TYPE ST_IOInputSimul :
STRUCT
	IxAru :BOOL;
END_STRUCT
END_TYPE

(* stored: Version 1.1.0.1, ProductVersion 3.1.4020.6
   DUT ST_IOInputSimul: Id {0eeda127-7f03-4f22-8390-7883b0f0db7e} *)
